FUNCTION F_AlarmPrioToText : ST_Text
VAR_INPUT
	ePriority : E_AlarmPriority;
END_VAR

			
CASE ePriority OF
	E_AlarmPriority.Error:
		F_AlarmPrioToText := Const.stTextListGlobal.stText_Error;
		
	E_AlarmPriority.Warning:
		F_AlarmPrioToText := Const.stTextListGlobal.stText_Warning;
		
	ELSE
		F_AlarmPrioToText := Const.stTextListGlobal.stText_Info;
	
END_CASE

END_FUNCTION

(* stored: Version 1.1.0.1, ProductVersion 3.1.4024.11
   POU F_AlarmPrioToText: Id {e8138bc9-9a54-4006-8af7-cf2d386958b2}, SpecialFunc None *)
